Universal Robots PolyScope program: programa1.urp

Program programa1 (installation=default directory=/ursim/programs createdIn=5.26.1 lastSavedIn=5.26.1 robotSerialNumber=20195599999)
Calibrated DH parameters: a=[0, -0.425, -0.3922, 0, 0, 0]; d=[0.1625, 0, 0, 0.1333, 0.0997, 0.0996]; alpha=[1.570796, 0, 0, 1.570796, -1.570796, 0]; deltaTheta=[0, 0, 0, 0, 0, 0]
InitVariablesNode
Robot Program (runOnlyOnce=true)
  Popup Message (haltProgram=false message=se va a simular la letra j inputType=Text)
  Script file /ursim/programs/letraJ1.script
    | movej(p[-0.225,-0.350,-0.050,0,3.1416,0], a=1.0, v=0.5)
    | movel(p[-0.300,-0.300,-0.100,0,3.1416,0], a=0.5, v=0.1)
    | movel(p[-0.300,-0.300,-0.150,0,3.1416,0], a=0.5, v=0.1)
    | movel(p[-0.240,-0.300,-0.150,0,3.1416,0], a=0.5, v=0.1)
    | movel(p[-0.260,-0.300,-0.150,0,3.1416,0], a=0.5, v=0.1)
    | movel(p[-0.260,-0.375,-0.150,0,3.1416,0], a=0.5, v=0.1)
    | movec(p[-0.280,-0.395,-0.150,0,3.1416,0], p[-0.300,-0.375,-0.150,0,3.1416,0], a=0.5, v=0.1)
    | movel(p[-0.300,-0.375,-0.100,0,3.1416,0], a=0.5, v=0.1)
  Popup Message (haltProgram=false message=simular la letra c inputType=Text)
  Script file /ursim/programs/letraC.script
    | movel(p[-0.150,-0.300,-0.100,0,3.1416,0], a=0.5, v=0.1)
    | movel(p[-0.150,-0.300,-0.150,0,3.1416,0], a=0.5, v=0.1)
    | movec(p[-0.200,-0.350,-0.150,0,3.1416,0], p[-0.150,-0.400,-0.150,0,3.1416,0], a=0.5, v=0.1)
    | movel(p[-0.150,-0.400,-0.100,0,3.1416,0], a=0.5, v=0.1)
  Popup Message (haltProgram=false message=se va a smilar la la letra j2 inputType=Text)
  Script file /ursim/programs/letraJ2.script
    | movel(p[-0.100,-0.300,-0.100,0,3.1416,0], a=0.5, v=0.1)
    | movel(p[-0.100,-0.300,-0.150,0,3.1416,0], a=0.5, v=0.1)
    | movel(p[-0.040,-0.300,-0.150,0,3.1416,0], a=0.5, v=0.1)
    | movel(p[-0.060,-0.300,-0.150,0,3.1416,0], a=0.5, v=0.1)
    | movel(p[-0.060,-0.375,-0.150,0,3.1416,0], a=0.5, v=0.1)
    | movec(p[-0.080,-0.395,-0.150,0,3.1416,0], p[-0.100,-0.375,-0.150,0,3.1416,0], a=0.5, v=0.1)
    | movel(p[-0.100,-0.375,-0.100,0,3.1416,0], a=0.5, v=0.1)
  Popup Message (haltProgram=false message=se va a simular la s inputType=Text)
  Script file /ursim/programs/letraS.script
    | movel(p[0.050,-0.300,-0.100,0,3.1416,0], a=0.5, v=0.1)
    | movel(p[0.050,-0.300,-0.150,0,3.1416,0], a=0.5, v=0.1)
    | movel(p[0.030,-0.300,-0.150,0,3.1416,0], a=0.5, v=0.1)
    | movec(p[0.005,-0.325,-0.150,0,3.1416,0], p[0.030,-0.350,-0.150,0,3.1416,0], a=0.5, v=0.1)
    | movec(p[0.055,-0.375,-0.150,0,3.1416,0], p[0.030,-0.400,-0.150,0,3.1416,0], a=0.5, v=0.1)
    | movel(p[0.010,-0.400,-0.150,0,3.1416,0], a=0.5, v=0.1)
    | movel(p[0.010,-0.400,-0.100,0,3.1416,0], a=0.5, v=0.1)
    | movej(p[-0.225,-0.350,-0.050,0,3.1416,0], a=1.0, v=0.5)
